   A_28_A408Z1O1.StFault := FALSE;
   A_28_A408Z1O1.StFalse := FALSE;
   A_28_A408Z1O1.spare0506 := FALSE;
   A_28_A408Z1O1.OutPausing := FALSE;
   A_28_A408Z1O1.OutAlarmNrLog := 0;
   A_28_A408Z1O1.Par.ParObjectNo := 1432;
   A_28_A408Z1O1.Par.ParMsgType := 7002;
   A_28_A408Z1O1.Par.ParHornCode := 9;
   A_28_A408Z1O1.Par.ParLogOff := FALSE;
   A_28_A408Z1O1.Par.ParManual := TRUE;
   A_28_A408Z1O1.Par.ParContinuous := TRUE;
   A_28_A408Z1O1.Par.ParPulse := FALSE;
   A_28_A408Z1O1.Par.ParPulsing := FALSE;
   A_28_A408Z1O1.Par.ParFilter := FALSE;
   A_28_A408Z1O1.Par.ParOnTime := 10;
   A_28_A408Z1O1.Par.ParOffTime := 0;
   A_28_A408Z1O1.Par.ParIdlingTime := 0;
   A_28_A408Z1O1.Par.ParDelayTime := 0;
   A_28_A408Z1O1.Par.OutTime := 0;
   A_28_A408Z1O1.Par.OutDelayTime := 0;
   A_28_A408Z1O1.Par.spare26 := 0;
   A_28_A408Z1O1.Par.spare28 := 0;
   A_28_A408Z1O1.Par.InOutManPulseLen := 0;
   A_28_A700Z1.StCode := 0;
   A_28_A700Z1.InMonTrue := FALSE;
   A_28_A700Z1.InMonFalse := FALSE;
   A_28_A700Z1.InPreAlarmTrue := FALSE;
   A_28_A700Z1.InPreAlarmFalse := FALSE;
   A_28_A700Z1.InStopTrueTime := FALSE;
   A_28_A700Z1.InStopFalseTime := FALSE;
   A_28_A700Z1.InpTrue := FALSE;
   A_28_A700Z1.InpFaultDev := FALSE;
   A_28_A700Z1.CmdRstTrueTime := FALSE;
   A_28_A700Z1.CmdRstFalseTime := FALSE;
   A_28_A700Z1.CmdRunTimeoutTime := FALSE;
   A_28_A700Z1.CmdFaultReset := FALSE;
   A_28_A700Z1.InLocal := FALSE;
   A_28_A700Z1.spare0305 := FALSE;
   A_28_A700Z1.InReport := FALSE;
   A_28_A700Z1.OutTimeoutTime := FALSE;
   A_28_A700Z1.InHWStop := FALSE;
   A_28_A700Z1.InDPFault := FALSE;
   A_28_A700Z1.OutPreAlarmTrue := FALSE;
   A_28_A700Z1.OutPreAlarmFalse := FALSE;
   A_28_A700Z1.OutFlagPos := FALSE;
   A_28_A700Z1.OutFlagNeg := FALSE;
   A_28_A700Z1.OutpFaultReset := FALSE;
   A_28_A700Z1.OutTrue := FALSE;
   A_28_A700Z1.StFalse := FALSE;
   A_28_A700Z1.StCtoTrue := FALSE;
   A_28_A700Z1.StTrue := FALSE;
   A_28_A700Z1.StCtoFalse := FALSE;
   A_28_A700Z1.StFault := FALSE;
   A_28_A700Z1.OutAlarmNrLog := 0;
   A_28_A700Z1.Par.ParObjectNo := 1433;
   A_28_A700Z1.Par.ParMsgType := 7147;
   A_28_A700Z1.Par.ParHornCode := 9;
   A_28_A700Z1.Par.ParLogOff := FALSE;
   A_28_A700Z1.Par.spare0401 := FALSE;
   A_28_A700Z1.Par.Par2WorkingCond := FALSE;
   A_28_A700Z1.Par.ParFaultRetry := FALSE;
   A_28_A700Z1.Par.ParBinLevel := FALSE;
   A_28_A700Z1.Par.ParDelayChange := 0;
   A_28_A700Z1.Par.ParDelayTrue := 10;
   A_28_A700Z1.Par.ParDelayFalse := 0;
   A_28_A700Z1.Par.ParTimeoutTrue := 0;
   A_28_A700Z1.Par.ParTimeoutFalse := 0;
   A_28_A700Z1.Par.OutMonTime := 0;
   A_28_A700Z1.Par.OutTransitionTime := 0;
   A_28_A700Z1.Par.OutMonTrue := FALSE;
   A_28_A700Z1.Par.OutMonFalse := FALSE;
   A_28_A700Z1.Par.OutFlagFaultDev := FALSE;
   A_28_A700Z1.Par.OutDelayTime := 0;
   A_28_A800Z1.StCode := 0;
   A_28_A800Z1.InMonTrue := FALSE;
   A_28_A800Z1.InMonFalse := FALSE;
   A_28_A800Z1.InPreAlarmTrue := FALSE;
   A_28_A800Z1.InPreAlarmFalse := FALSE;
   A_28_A800Z1.InStopTrueTime := FALSE;
   A_28_A800Z1.InStopFalseTime := FALSE;
   A_28_A800Z1.InpTrue := FALSE;
   A_28_A800Z1.InpFaultDev := FALSE;
   A_28_A800Z1.CmdRstTrueTime := FALSE;
   A_28_A800Z1.CmdRstFalseTime := FALSE;
   A_28_A800Z1.CmdRunTimeoutTime := FALSE;
   A_28_A800Z1.CmdFaultReset := FALSE;
   A_28_A800Z1.InLocal := FALSE;
   A_28_A800Z1.spare0305 := FALSE;
   A_28_A800Z1.InReport := FALSE;
   A_28_A800Z1.OutTimeoutTime := FALSE;
   A_28_A800Z1.InHWStop := FALSE;
   A_28_A800Z1.InDPFault := FALSE;
   A_28_A800Z1.OutPreAlarmTrue := FALSE;
   A_28_A800Z1.OutPreAlarmFalse := FALSE;
   A_28_A800Z1.OutFlagPos := FALSE;
   A_28_A800Z1.OutFlagNeg := FALSE;
   A_28_A800Z1.OutpFaultReset := FALSE;
   A_28_A800Z1.OutTrue := FALSE;
   A_28_A800Z1.StFalse := FALSE;
   A_28_A800Z1.StCtoTrue := FALSE;
   A_28_A800Z1.StTrue := FALSE;
   A_28_A800Z1.StCtoFalse := FALSE;
   A_28_A800Z1.StFault := FALSE;
   A_28_A800Z1.OutAlarmNrLog := 0;
   A_28_A800Z1.Par.ParObjectNo := 1434;
   A_28_A800Z1.Par.ParMsgType := 7147;
   A_28_A800Z1.Par.ParHornCode := 9;
   A_28_A800Z1.Par.ParLogOff := FALSE;
   A_28_A800Z1.Par.spare0401 := FALSE;
   A_28_A800Z1.Par.Par2WorkingCond := FALSE;
   A_28_A800Z1.Par.ParFaultRetry := FALSE;
   A_28_A800Z1.Par.ParBinLevel := FALSE;
   A_28_A800Z1.Par.ParDelayChange := 0;
   A_28_A800Z1.Par.ParDelayTrue := 10;
   A_28_A800Z1.Par.ParDelayFalse := 0;
   A_28_A800Z1.Par.ParTimeoutTrue := 0;
   A_28_A800Z1.Par.ParTimeoutFalse := 0;
   A_28_A800Z1.Par.OutMonTime := 0;
   A_28_A800Z1.Par.OutTransitionTime := 0;
   A_28_A800Z1.Par.OutMonTrue := FALSE;
   A_28_A800Z1.Par.OutMonFalse := FALSE;
   A_28_A800Z1.Par.OutFlagFaultDev := FALSE;
   A_28_A800Z1.Par.OutDelayTime := 0;
//Parameter =A-28-A106Z1 : EMERGENCY STOP FROM +C27
      #A_28_A106Z1.Par.ParObjectNo                             :=1435;
      #A_28_A106Z1.Par.ParMsgType                              :=7171;
      #A_28_A106Z1.Par.ParHornCode                             :=2;
      #A_28_A106Z1.Par.ParDelayChange                          :=0;
      #A_28_A106Z1.Par.ParDelayTrue                            :=10;
      #A_28_A106Z1.Par.ParDelayFalse                           :=0;
      #A_28_A106Z1.Par.ParTimeoutTrue                          :=0;
      #A_28_A106Z1.Par.ParTimeoutFalse                         :=0;
      #A_28_A106Z1.Par.ParLogOff                               :=False;
      #A_28_A106Z1.Par.Par2WorkingCond                         :=False;
      #A_28_A106Z1.Par.ParFaultRetry                           :=False;
      #A_28_A106Z1.Par.ParBinLevel                             :=False;
//
//
END_DATA_BLOCK

